// TIA Portal V18 export
FUNCTION_BLOCK "MU_Torq"   // FB32, LAD
TITLE = MU Torq
{ S7_Optimized_Access := 'TRUE' }
// Written BY Kristopher Gimenez Feb 3,2023
// This block is used to control the TD MU Torq mode
// stored: AutoNumber false, MemoryReserve 100, SetENOAutomatically false
   VAR_INPUT
      Start : Bool;
   END_VAR
   VAR_OUTPUT
      FlowFwdmAOut : Real;
      TorqmAOut : Real;
      EnableP1 : Bool;
      EnableP2 { ExternalWritable := 'False'} : Bool;
      TorqEn : Bool;
      MUSeqRunning : Bool;
   END_VAR
   VAR
      MUspeed : Real;
      PumpToggle : Bool;   // Bit will toggle each make up sequence to choose which pump to stroke. 0 = P1, 1 = P2
      AutoMUComplete : Bool;
      RampDown : Bool;   // Bit to know system need to ramp down
      RampDownComplete : Bool;   // Indicates Ramp Down completed
      MUComplete_TON { S7_SetPoint := 'True'} : TON_TIME;
      TorqUserSetmA : Real;
      AutoMUInc_TON { S7_SetPoint := 'True'} : TON_TIME;
      Torq_Ramp { S7_SetPoint := 'True'} : RampFunction;
      Flow_Ramp { S7_SetPoint := 'True'} : RampFunction;
      TorqRampInmA { S7_SetPoint := 'True'} : Real;   // Value assigned to ramp fucntion to get ramped output
      FlowRampInmA : Real;   // Value assigned to ramp fucntion to get ramped ouput
      MUSeqRunLast : Bool;
   END_VAR
   VAR_TEMP
      TorqPSITemp : Real;
      tempReal : Real;
      toggleTemp : Bool;
   END_VAR
   VAR_TEMP   // added for the SCL form of the ladder/FBD networks
      _w1 : Bool;
      _w2 : Bool;
      _w3 : Bool;
      _w4 : Bool;
      _w5 : Bool;
      _w6 : Bool;
      _w7 : Bool;
   END_VAR
BEGIN

REGION Network 1: Set Running
   // Set running bit and trigger resets when starting a MU sequence
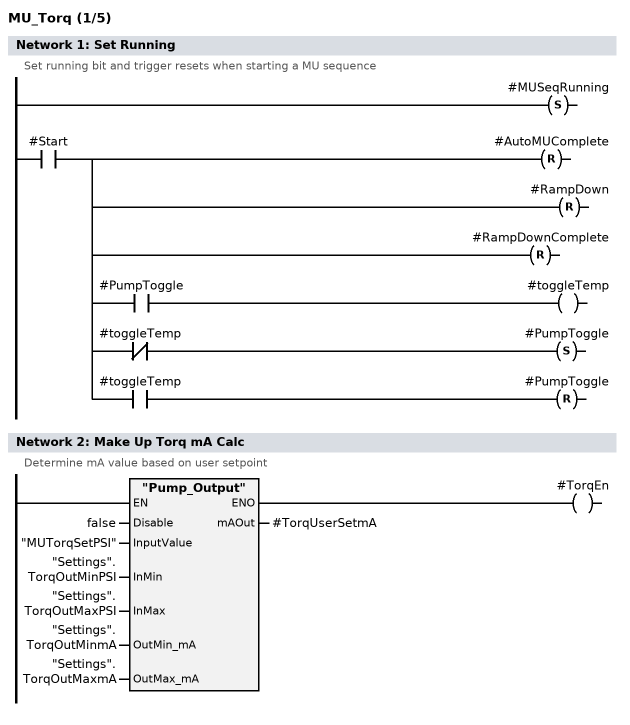
   RUNG wire#powerrail
      S_Coil( #MUSeqRunning )
   END_RUNG
   RUNG wire#powerrail
      Contact( #Start )
      wire#w1
      R_Coil( #AutoMUComplete )
   END_RUNG
   RUNG wire#w1
      R_Coil( #RampDown )
   END_RUNG
   RUNG wire#w1
      R_Coil( #RampDownComplete )
   END_RUNG
   RUNG wire#w1
      Contact( #PumpToggle )
      Coil( #toggleTemp )
   END_RUNG
   RUNG wire#w1
      I_Contact( #toggleTemp )
      S_Coil( #PumpToggle )
   END_RUNG
   RUNG wire#w1
      Contact( #toggleTemp )
      R_Coil( #PumpToggle )
   END_RUNG
   // the same network as SCL:
   #MUSeqRunning := TRUE;
   IF #Start THEN
       #AutoMUComplete := FALSE;
       #RampDown := FALSE;
       #RampDownComplete := FALSE;
   END_IF;
   #toggleTemp := #Start AND #PumpToggle;
   IF #Start AND NOT #toggleTemp THEN #PumpToggle := TRUE; END_IF;
   IF #Start AND #toggleTemp THEN #PumpToggle := FALSE; END_IF;
END_REGION

REGION Network 2: Make Up Torq mA Calc
   // Determine mA value based on user setpoint
   RUNG wire#powerrail
      "Pump_Output"(Disable := false, InputValue := "MUTorqSetPSI", InMin := "Settings".TorqOutMinPSI, InMax := "Settings".TorqOutMaxPSI, OutMin_mA := "Settings".TorqOutMinmA, OutMax_mA := "Settings".TorqOutMaxmA, mAOut => #TorqUserSetmA)
      Coil( #TorqEn )
   END_RUNG
   // the same network as SCL:
   "Pump_Output"(Disable := false,
                 InputValue := "MUTorqSetPSI",
                 InMin := "Settings".TorqOutMinPSI,
                 InMax := "Settings".TorqOutMaxPSI,
                 OutMin_mA := "Settings".TorqOutMinmA,
                 OutMax_mA := "Settings".TorqOutMaxmA,
                 mAOut => #TorqUserSetmA,
                 ENO => #_w1);
   #TorqEn := #_w1;
END_REGION

REGION Network 3: Mu torque speed setting based on torque setpoint
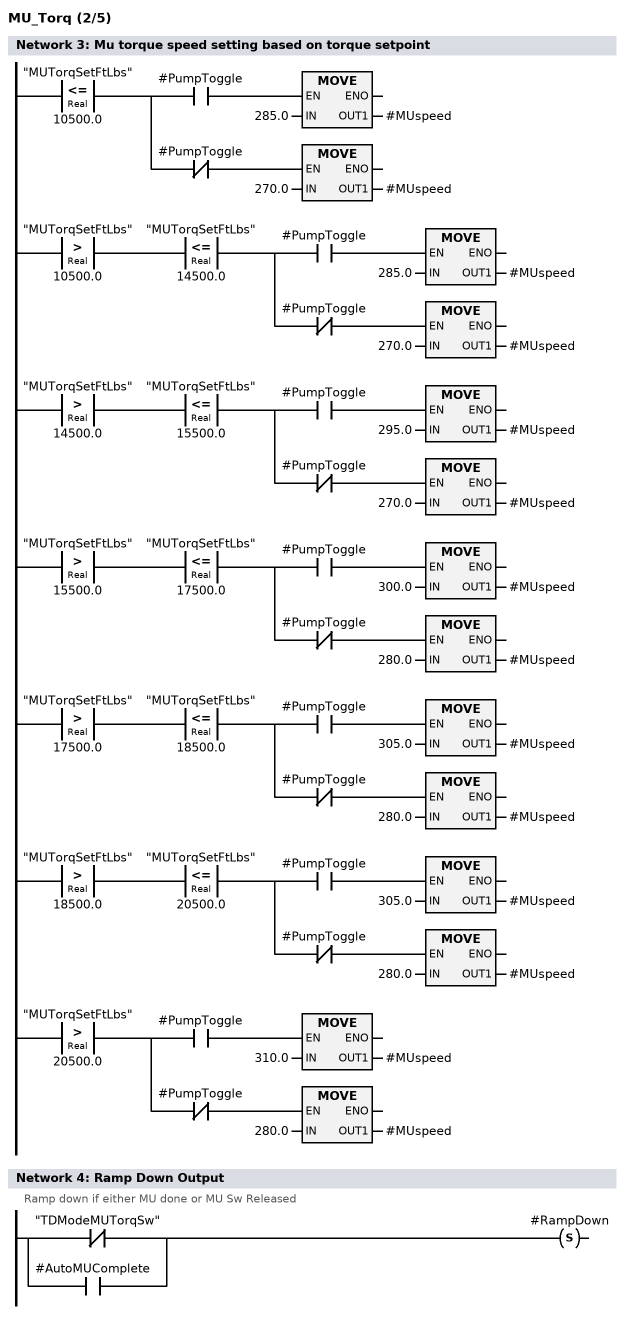
   RUNG wire#powerrail
      { S7_Templates := "SrcType := Real" } LE_Contact(in1 := "MUTorqSetFtLbs", in2 := 10500.0)
      wire#w1
      Contact( #PumpToggle )
      Move(in := 285.0, out1 => #MUspeed)
   END_RUNG
   RUNG wire#w1
      I_Contact( #PumpToggle )
      Move(in := 270.0, out1 => #MUspeed)
   END_RUNG
   RUNG wire#powerrail
      { S7_Templates := "SrcType := Real" } GT_Contact(in1 := "MUTorqSetFtLbs", in2 := 10500.0)
      { S7_Templates := "SrcType := Real" } LE_Contact(in1 := "MUTorqSetFtLbs", in2 := 14500.0)
      wire#w2
      Contact( #PumpToggle )
      Move(in := 285.0, out1 => #MUspeed)
   END_RUNG
   RUNG wire#w2
      I_Contact( #PumpToggle )
      Move(in := 270.0, out1 => #MUspeed)
   END_RUNG
   RUNG wire#powerrail
      { S7_Templates := "SrcType := Real" } GT_Contact(in1 := "MUTorqSetFtLbs", in2 := 14500.0)
      { S7_Templates := "SrcType := Real" } LE_Contact(in1 := "MUTorqSetFtLbs", in2 := 15500.0)
      wire#w3
      Contact( #PumpToggle )
      Move(in := 295.0, out1 => #MUspeed)
   END_RUNG
   RUNG wire#w3
      I_Contact( #PumpToggle )
      Move(in := 270.0, out1 => #MUspeed)
   END_RUNG
   RUNG wire#powerrail
      { S7_Templates := "SrcType := Real" } GT_Contact(in1 := "MUTorqSetFtLbs", in2 := 15500.0)
      { S7_Templates := "SrcType := Real" } LE_Contact(in1 := "MUTorqSetFtLbs", in2 := 17500.0)
      wire#w4
      Contact( #PumpToggle )
      Move(in := 300.0, out1 => #MUspeed)
   END_RUNG
   RUNG wire#w4
      I_Contact( #PumpToggle )
      Move(in := 280.0, out1 => #MUspeed)
   END_RUNG
   RUNG wire#powerrail
      { S7_Templates := "SrcType := Real" } GT_Contact(in1 := "MUTorqSetFtLbs", in2 := 17500.0)
      { S7_Templates := "SrcType := Real" } LE_Contact(in1 := "MUTorqSetFtLbs", in2 := 18500.0)
      wire#w5
      Contact( #PumpToggle )
      Move(in := 305.0, out1 => #MUspeed)
   END_RUNG
   RUNG wire#w5
      I_Contact( #PumpToggle )
      Move(in := 280.0, out1 => #MUspeed)
   END_RUNG
   RUNG wire#powerrail
      { S7_Templates := "SrcType := Real" } GT_Contact(in1 := "MUTorqSetFtLbs", in2 := 18500.0)
      { S7_Templates := "SrcType := Real" } LE_Contact(in1 := "MUTorqSetFtLbs", in2 := 20500.0)
      wire#w6
      Contact( #PumpToggle )
      Move(in := 305.0, out1 => #MUspeed)
   END_RUNG
   RUNG wire#w6
      I_Contact( #PumpToggle )
      Move(in := 280.0, out1 => #MUspeed)
   END_RUNG
   RUNG wire#powerrail
      { S7_Templates := "SrcType := Real" } GT_Contact(in1 := "MUTorqSetFtLbs", in2 := 20500.0)
      wire#w7
      Contact( #PumpToggle )
      Move(in := 310.0, out1 => #MUspeed)
   END_RUNG
   RUNG wire#w7
      I_Contact( #PumpToggle )
      Move(in := 280.0, out1 => #MUspeed)
   END_RUNG
   // the same network as SCL:
   #_w1 := "MUTorqSetFtLbs" <= 10500.0;
   IF #_w1 AND #PumpToggle THEN #MUspeed := 285.0; END_IF;
   IF #_w1 AND NOT #PumpToggle THEN #MUspeed := 270.0; END_IF;
   #_w2 := ("MUTorqSetFtLbs" > 10500.0) AND ("MUTorqSetFtLbs" <= 14500.0);
   IF #_w2 AND #PumpToggle THEN #MUspeed := 285.0; END_IF;
   IF #_w2 AND NOT #PumpToggle THEN #MUspeed := 270.0; END_IF;
   #_w3 := ("MUTorqSetFtLbs" > 14500.0) AND ("MUTorqSetFtLbs" <= 15500.0);
   IF #_w3 AND #PumpToggle THEN #MUspeed := 295.0; END_IF;
   IF #_w3 AND NOT #PumpToggle THEN #MUspeed := 270.0; END_IF;
   #_w4 := ("MUTorqSetFtLbs" > 15500.0) AND ("MUTorqSetFtLbs" <= 17500.0);
   IF #_w4 AND #PumpToggle THEN #MUspeed := 300.0; END_IF;
   IF #_w4 AND NOT #PumpToggle THEN #MUspeed := 280.0; END_IF;
   #_w5 := ("MUTorqSetFtLbs" > 17500.0) AND ("MUTorqSetFtLbs" <= 18500.0);
   IF #_w5 AND #PumpToggle THEN #MUspeed := 305.0; END_IF;
   IF #_w5 AND NOT #PumpToggle THEN #MUspeed := 280.0; END_IF;
   #_w6 := ("MUTorqSetFtLbs" > 18500.0) AND ("MUTorqSetFtLbs" <= 20500.0);
   IF #_w6 AND #PumpToggle THEN #MUspeed := 305.0; END_IF;
   IF #_w6 AND NOT #PumpToggle THEN #MUspeed := 280.0; END_IF;
   #_w7 := "MUTorqSetFtLbs" > 20500.0;
   IF #_w7 AND #PumpToggle THEN #MUspeed := 310.0; END_IF;
   IF #_w7 AND NOT #PumpToggle THEN #MUspeed := 280.0; END_IF;
END_REGION

REGION Network 4: Ramp Down Output
   // Ramp down if either MU done or MU Sw Released
   RUNG wire#powerrail
      I_Contact( "TDModeMUTorqSw" )
      wire#w1
      S_Coil( #RampDown )
   END_RUNG
   RUNG wire#powerrail
      Contact( #AutoMUComplete )
   END_RUNG wire#w1
   // the same network as SCL:
   IF NOT "TDModeMUTorqSw" OR #AutoMUComplete THEN #RampDown := TRUE; END_IF;
END_REGION

REGION Network 5: Assign Torq Ramp Parameters
   // Set Torq Ramp settings as needed. If Transducer faulted use default values. If no TX fault, in Auto Mode set value based on Torq feedback
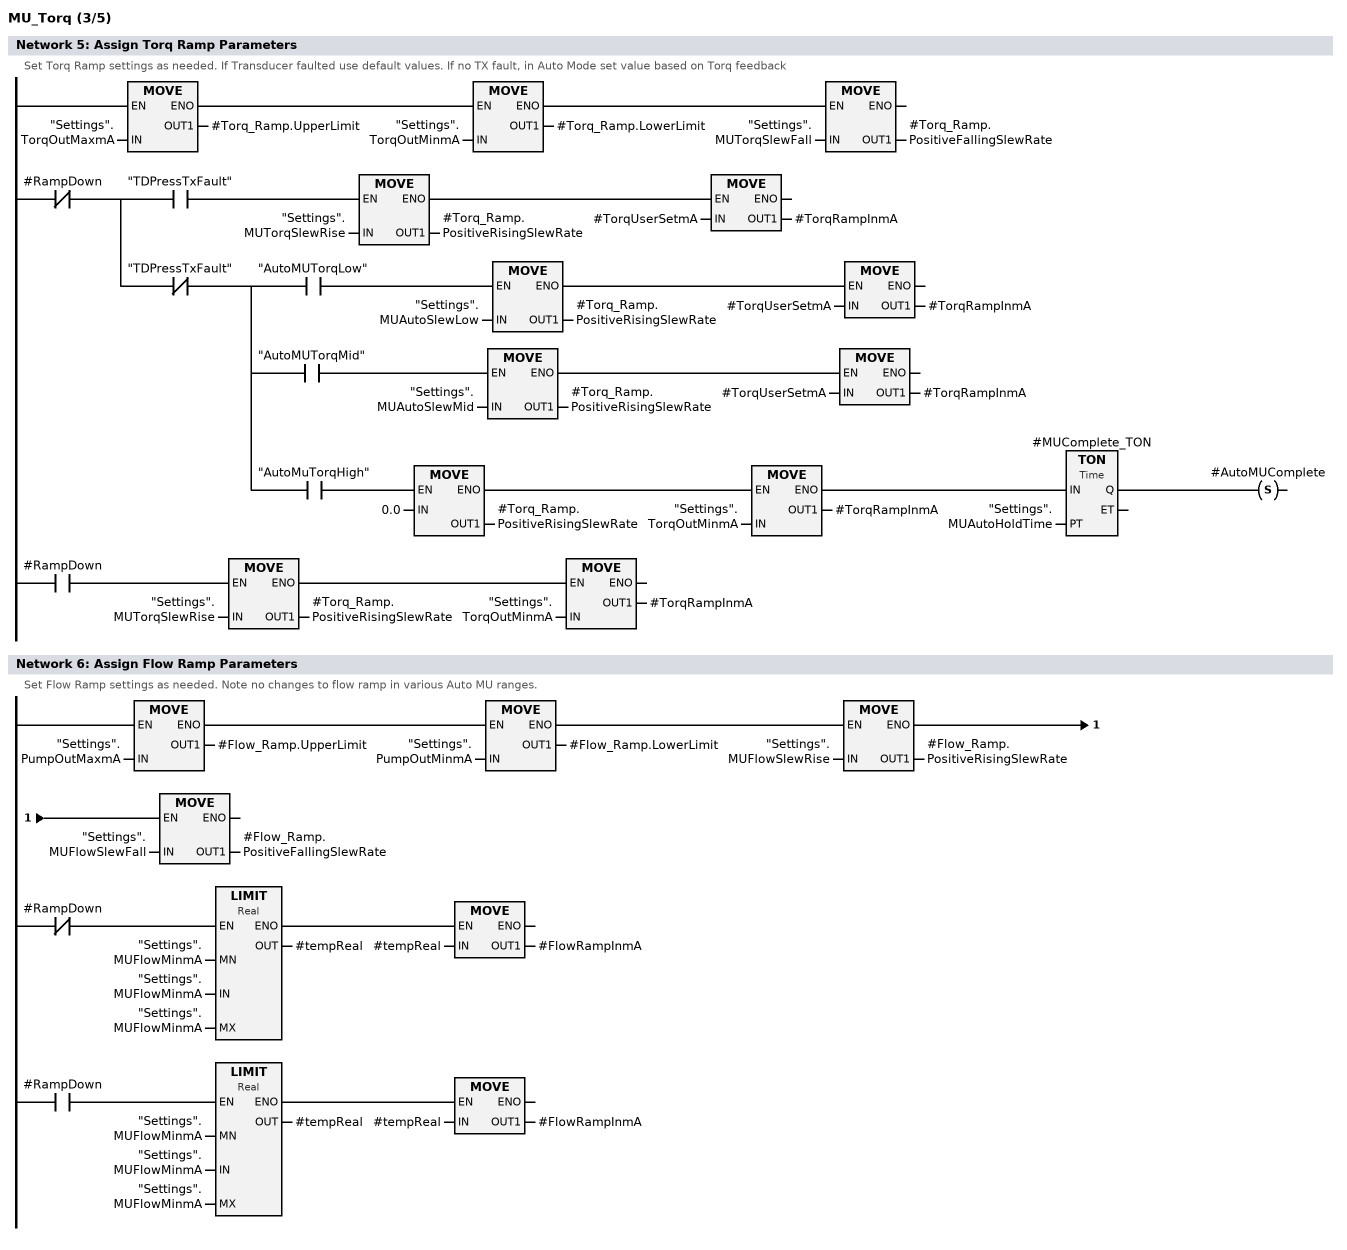
   RUNG wire#powerrail
      Move(in := "Settings".TorqOutMaxmA, out1 => #Torq_Ramp.UpperLimit)
      Move(in := "Settings".TorqOutMinmA, out1 => #Torq_Ramp.LowerLimit)
      Move(in := "Settings".MUTorqSlewFall, out1 => #Torq_Ramp.PositiveFallingSlewRate)
   END_RUNG
   RUNG wire#powerrail
      I_Contact( #RampDown )
      wire#w1
      Contact( "TDPressTxFault" )
      Move(in := "Settings".MUTorqSlewRise, out1 => #Torq_Ramp.PositiveRisingSlewRate)
      Move(in := #TorqUserSetmA, out1 => #TorqRampInmA)
   END_RUNG
   RUNG wire#w1
      I_Contact( "TDPressTxFault" )
      wire#w2
      Contact( "AutoMUTorqLow" )
      Move(in := "Settings".MUAutoSlewLow, out1 => #Torq_Ramp.PositiveRisingSlewRate)
      Move(in := #TorqUserSetmA, out1 => #TorqRampInmA)
   END_RUNG
   RUNG wire#w2
      Contact( "AutoMUTorqMid" )
      Move(in := "Settings".MUAutoSlewMid, out1 => #Torq_Ramp.PositiveRisingSlewRate)
      Move(in := #TorqUserSetmA, out1 => #TorqRampInmA)
   END_RUNG
   RUNG wire#w2
      Contact( "AutoMuTorqHigh" )
      Move(in := 0.0, out1 => #Torq_Ramp.PositiveRisingSlewRate)
      Move(in := "Settings".TorqOutMinmA, out1 => #TorqRampInmA)
      { S7_Templates := "time_type := Time" } #MUComplete_TON.TON(pt := "Settings".MUAutoHoldTime, et =>)
      S_Coil( #AutoMUComplete )
   END_RUNG
   RUNG wire#powerrail
      Contact( #RampDown )
      Move(in := "Settings".MUTorqSlewRise, out1 => #Torq_Ramp.PositiveRisingSlewRate)
      Move(in := "Settings".TorqOutMinmA, out1 => #TorqRampInmA)
   END_RUNG
   // the same network as SCL:
   #Torq_Ramp.UpperLimit := "Settings".TorqOutMaxmA;
   #Torq_Ramp.LowerLimit := "Settings".TorqOutMinmA;
   #Torq_Ramp.PositiveFallingSlewRate := "Settings".MUTorqSlewFall;
   IF NOT #RampDown AND "TDPressTxFault" THEN
       #Torq_Ramp.PositiveRisingSlewRate := "Settings".MUTorqSlewRise;
       #TorqRampInmA := #TorqUserSetmA;
   END_IF;
   #_w1 := NOT #RampDown AND NOT "TDPressTxFault";
   IF #_w1 AND "AutoMUTorqLow" THEN
       #Torq_Ramp.PositiveRisingSlewRate := "Settings".MUAutoSlewLow;
       #TorqRampInmA := #TorqUserSetmA;
   END_IF;
   IF #_w1 AND "AutoMUTorqMid" THEN
       #Torq_Ramp.PositiveRisingSlewRate := "Settings".MUAutoSlewMid;
       #TorqRampInmA := #TorqUserSetmA;
   END_IF;
   #_w2 := #_w1 AND "AutoMuTorqHigh";
   IF #_w2 THEN
       #Torq_Ramp.PositiveRisingSlewRate := 0.0;
       #TorqRampInmA := "Settings".TorqOutMinmA;
   END_IF;
   #MUComplete_TON(IN := #_w2, PT := "Settings".MUAutoHoldTime);   // TON
   IF #MUComplete_TON.Q THEN #AutoMUComplete := TRUE; END_IF;
   IF #RampDown THEN
       #Torq_Ramp.PositiveRisingSlewRate := "Settings".MUTorqSlewRise;
       #TorqRampInmA := "Settings".TorqOutMinmA;
   END_IF;
END_REGION

REGION Network 6: Assign Flow Ramp Parameters
   // Set Flow Ramp settings as needed. Note no changes to flow ramp in various Auto MU ranges.
   RUNG wire#powerrail
      Move(in := "Settings".PumpOutMaxmA, out1 => #Flow_Ramp.UpperLimit)
      Move(in := "Settings".PumpOutMinmA, out1 => #Flow_Ramp.LowerLimit)
      Move(in := "Settings".MUFlowSlewRise, out1 => #Flow_Ramp.PositiveRisingSlewRate)
      Move(in := "Settings".MUFlowSlewFall, out1 => #Flow_Ramp.PositiveFallingSlewRate)
   END_RUNG
   RUNG wire#powerrail
      I_Contact( #RampDown )
      { S7_Templates := "value_type := Real" } Limit(mn := "Settings".MUFlowMinmA, in := "Settings".MUFlowMinmA, mx := "Settings".MUFlowMinmA, out => #tempReal)
      Move(in := #tempReal, out1 => #FlowRampInmA)
   END_RUNG
   RUNG wire#powerrail
      Contact( #RampDown )
      { S7_Templates := "value_type := Real" } Limit(mn := "Settings".MUFlowMinmA, in := "Settings".MUFlowMinmA, mx := "Settings".MUFlowMinmA, out => #tempReal)
      Move(in := #tempReal, out1 => #FlowRampInmA)
   END_RUNG
   // the same network as SCL:
   #Flow_Ramp.UpperLimit := "Settings".PumpOutMaxmA;
   #Flow_Ramp.LowerLimit := "Settings".PumpOutMinmA;
   #Flow_Ramp.PositiveRisingSlewRate := "Settings".MUFlowSlewRise;
   #Flow_Ramp.PositiveFallingSlewRate := "Settings".MUFlowSlewFall;
   IF NOT #RampDown THEN
       #tempReal := LIMIT(MN := "Settings".MUFlowMinmA, IN := "Settings".MUFlowMinmA, MX := "Settings".MUFlowMinmA);
       #FlowRampInmA := #tempReal;
   END_IF;
   IF #RampDown THEN
       #tempReal := LIMIT(MN := "Settings".MUFlowMinmA, IN := "Settings".MUFlowMinmA, MX := "Settings".MUFlowMinmA);
       #FlowRampInmA := #tempReal;
   END_IF;
END_REGION

REGION Network 7: Ramp mA Signals
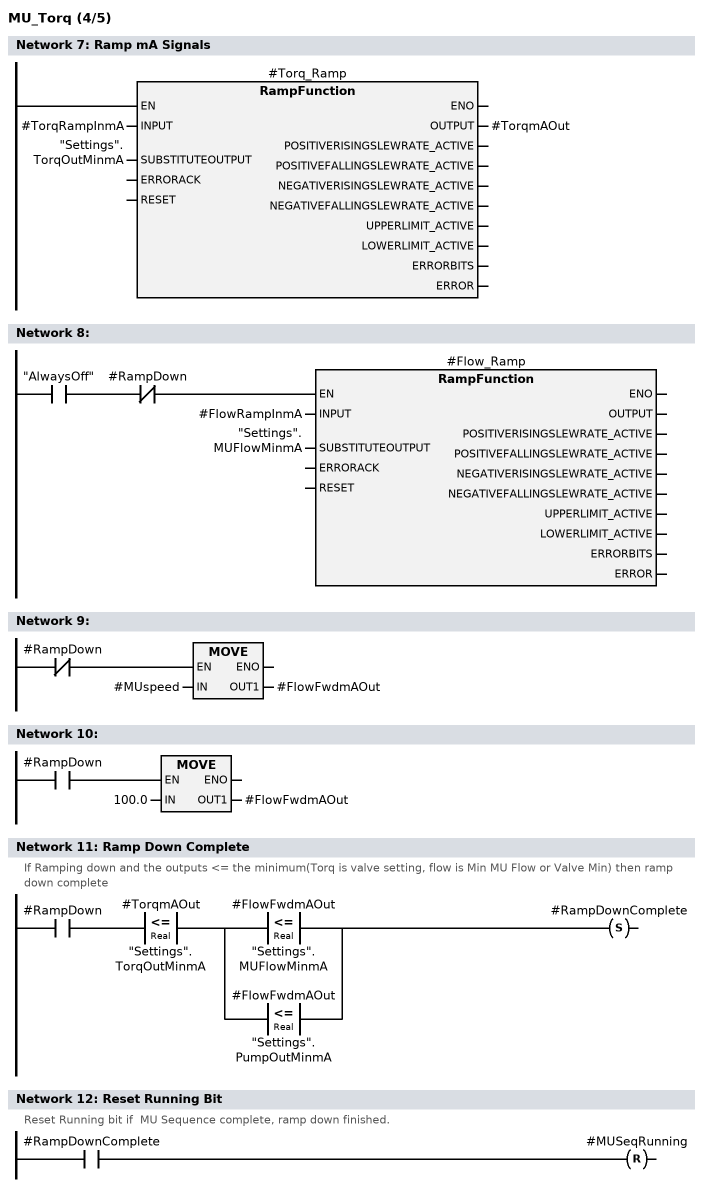
   RUNG wire#powerrail
      #Torq_Ramp.RampFunction(Input := #TorqRampInmA, SubstituteOutput := "Settings".TorqOutMinmA, ErrorAck :=, Reset :=, Output => #TorqmAOut, PositiveRisingSlewRate_Active =>, PositiveFallingSlewRate_Active =>, NegativeRisingSlewRate_Active =>, NegativeFallingSlewRate_Active =>, UpperLimit_Active =>, LowerLimit_Active =>, ErrorBits =>, Error =>)
   END_RUNG
   // the same network as SCL:
   #Torq_Ramp(Input := #TorqRampInmA, SubstituteOutput := "Settings".TorqOutMinmA, Output => #TorqmAOut);   // RampFunction
END_REGION

REGION Network 8
   RUNG wire#powerrail
      Contact( "AlwaysOff" )
      I_Contact( #RampDown )
      #Flow_Ramp.RampFunction(Input := #FlowRampInmA, SubstituteOutput := "Settings".MUFlowMinmA, ErrorAck :=, Reset :=, Output =>, PositiveRisingSlewRate_Active =>, PositiveFallingSlewRate_Active =>, NegativeRisingSlewRate_Active =>, NegativeFallingSlewRate_Active =>, UpperLimit_Active =>, LowerLimit_Active =>, ErrorBits =>, Error =>)
   END_RUNG
   // the same network as SCL:
   IF "AlwaysOff" AND NOT #RampDown THEN
       #Flow_Ramp(Input := #FlowRampInmA, SubstituteOutput := "Settings".MUFlowMinmA);   // RampFunction
   END_IF;
END_REGION

REGION Network 9
   RUNG wire#powerrail
      I_Contact( #RampDown )
      Move(in := #MUspeed, out1 => #FlowFwdmAOut)
   END_RUNG
   // the same network as SCL:
   IF NOT #RampDown THEN #FlowFwdmAOut := #MUspeed; END_IF;
END_REGION

REGION Network 10
   RUNG wire#powerrail
      Contact( #RampDown )
      Move(in := 100.0, out1 => #FlowFwdmAOut)
   END_RUNG
   // the same network as SCL:
   IF #RampDown THEN #FlowFwdmAOut := 100.0; END_IF;
END_REGION

REGION Network 11: Ramp Down Complete
   // If Ramping down and the outputs <= the minimum(Torq is valve setting, flow is Min MU Flow or Valve Min) then ramp down complete
   RUNG wire#powerrail
      Contact( #RampDown )
      { S7_Templates := "SrcType := Real" } LE_Contact(in1 := #TorqmAOut, in2 := "Settings".TorqOutMinmA)
      wire#w1
      { S7_Templates := "SrcType := Real" } LE_Contact(in1 := #FlowFwdmAOut, in2 := "Settings".MUFlowMinmA)
      wire#w2
      S_Coil( #RampDownComplete )
   END_RUNG
   RUNG wire#w1
      { S7_Templates := "SrcType := Real" } LE_Contact(in1 := #FlowFwdmAOut, in2 := "Settings".PumpOutMinmA)
   END_RUNG wire#w2
   // the same network as SCL:
   IF #RampDown AND (#TorqmAOut <= "Settings".TorqOutMinmA) AND ((#FlowFwdmAOut <= "Settings".MUFlowMinmA) OR (#FlowFwdmAOut <= "Settings".PumpOutMinmA)) THEN
       #RampDownComplete := TRUE;
   END_IF;
END_REGION

REGION Network 12: Reset Running Bit
   // Reset Running bit if  MU Sequence complete, ramp down finished.
   RUNG wire#powerrail
      Contact( #RampDownComplete )
      R_Coil( #MUSeqRunning )
   END_RUNG
   // the same network as SCL:
   IF #RampDownComplete THEN #MUSeqRunning := FALSE; END_IF;
END_REGION

REGION Network 13: Set Outputs
   // Torq always enabled in MU mode. Pumps alternate
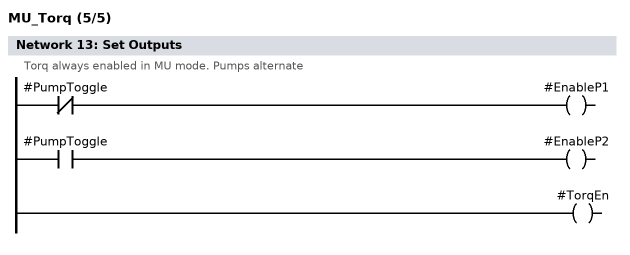
   RUNG wire#powerrail
      I_Contact( #PumpToggle )
      Coil( #EnableP1 )
   END_RUNG
   RUNG wire#powerrail
      Contact( #PumpToggle )
      Coil( #EnableP2 )
   END_RUNG
   RUNG wire#powerrail
      Coil( #TorqEn )
   END_RUNG
   // the same network as SCL:
   #EnableP1 := NOT #PumpToggle;
   #EnableP2 := #PumpToggle;
   #TorqEn := TRUE;
END_REGION
END_FUNCTION_BLOCK
